{attribute 'qualified_only'}
VAR_GLOBAL CONSTANT
	cIPAddr 			: STRING(15) := '169.254.222.244' ;
	cTCPPort			: UINT :=502;
	cUnitID				: BYTE :=255;
END_VAR

(* stored: Version 1.1.0.1, ProductVersion 3.1.4024.11
   GVL GCL_ModbusTcp: Id {ee2808e3-834e-4de2-895c-a020319decca} *)
